// TIA Portal project "TankFillingSystemSim" (V15)
// simulation of tank filling system

(* hardware
DEVICE "S7-1200 station_1"  S7-1200 Station
   slot 0: "Rack_0"  S7-1200 Rack  Rack  V1.0
   slot 1: "Filling System Controller"  CPU 1214C DC/DC/DC  6ES7 214-1AG40-0XB0  V4.2
   slot 3: "AQ 1x12BIT_1"  AQ1 signal board  6ES7 232-4HA30-0XB0  V1.0
   slot 101: "CM 1243-5"  CM 1243-5  6GK7 243-5DX30-0XE0  V1.3
   slot 102: "CM 1241 (RS485)_1"  CM 1241 (RS485)  6ES7 241-1CH30-0XB0  V1.0
*)

// ===== PLC "Filling System Controller"  CPU 1214C DC/DC/DC =====

VAR_GLOBAL   // PLC tag table "Default tag table"
   ""START"" AT %I0.0 : Bool;
   ""Bottom_Sensor1"" AT %I0.1 : Bool;
   ""Top_Sensor1"" AT %I0.2 : Bool;
   ""Confirm"" AT %I0.6 : Bool;
   ""Valve_Control"" AT %I0.3 : Bool;
   ""STOP"" AT %I0.7 : Bool;
   ""Tank1_Low_Level"" AT %Q0.0 : Bool;
   ""Tank1_Medium_Level"" AT %Q0.1 : Bool;
   ""Tank1_High_Level"" AT %Q0.2 : Bool;
   ""Tank1_Malfunction"" AT %Q0.3 : Bool;
   ""Valve_Status"" AT %Q0.4 : Bool;
   ""Pump_Status"" AT %Q0.5 : Bool;
END_VAR